KUKA KRL program: ToolRackClose.src

&ACCESS RVO6
&REL 8
&PARAM EDITMASK = *
&PARAM TEMPLATE = C:\KRC\Roboter\Template\vorgabe
DEF ToolRackClose( )
;FOLD INI;%{PE}
  ;FOLD BASISTECH INI
    GLOBAL INTERRUPT DECL 3 WHEN $STOPMESS==TRUE DO IR_STOPM ( )
    INTERRUPT ON 3
    BAS (#INITMOV,0 )
  ;ENDFOLD (BASISTECH INI)
  ;FOLD USER INI
    ;Make your modifications here

  ;ENDFOLD (USER INI)
;ENDFOLD (INI)

;************************************************
;              CNC Robotics Ltd
;              www.cncrobotics.co.uk
;************************************************
;     Contact: helpdesk@cncrobotics.co.uk
;     Date: 25/09/23
;     Version: 1.12.38
;     Date: 25/09/23
;     Version: 1.13.46
;************************************************
; Description: Close tool rack lid.
;************************************************


oOpenToolRack = FALSE ;Cancel tool rack open

WAIT SEC 0.25 ;Time delay

oCloseToolRack = TRUE ;Signal to close tool rack lid

WAIT FOR (iToolRackClosed) ;Wait for tool rack closed signal

END
